(* CoDeSys 2.3 export: ST_ISSUE94.EXP *)

(* Data type *)
TYPE ST_Issue94 :
STRUCT
	BoolValue 	: BOOL := TRUE;
	ArrayValue 	:  ARRAY [0..1] OF ST_Issue94_Byte := (ByteValue := 1), (ByteValue := 2);
END_STRUCT
END_TYPE
